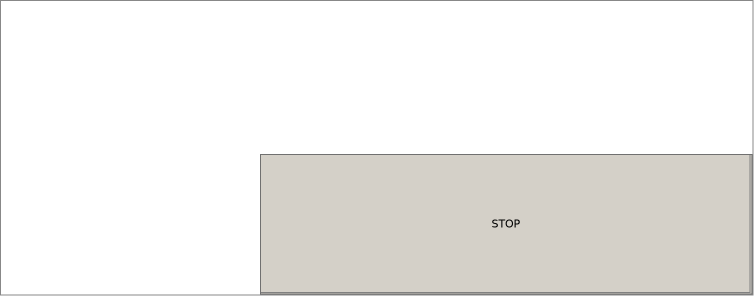
VISUALIZATION STOP  // 754x296
    Button (260,154 492x140), "STOP"
END_VISUALIZATION

(* stored: Version 1.1.0.1, ProductVersion 3.1.4024.2
   Visu STOP: Id {75d434c3-a557-4e40-af88-d7e84d4bfa3f} *)
